Yaskawa INFORM job: turntable_planes_program.JBI

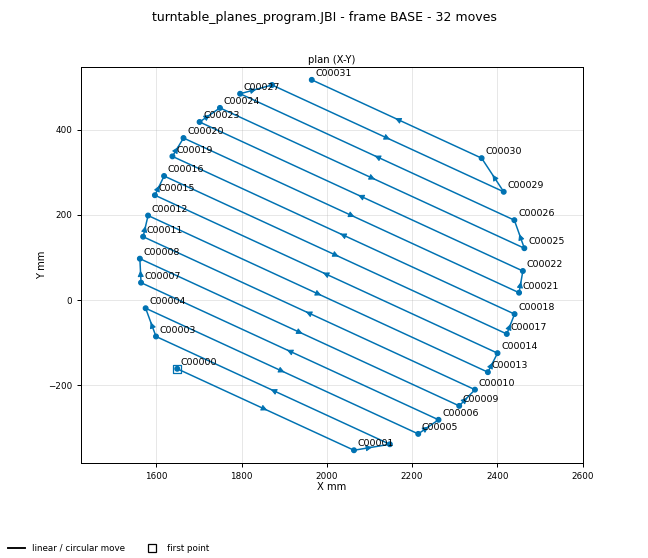
[picture p0: tool path of turntable_planes_program.JBI in frame BASE, 32 of 34 moves have a stored position in this frame; points joined in program order, loops and branches not executed]
/JOB
//NAME turntable_planes_program
//POS
///NPOS 32,0,32,0,0,0
///TOOL 0
///POSTYPE BASE
///RECTAN
///RCONF 0,0,0,0,0,0,0,0,0,0,0,0,0,0,0,0,0,0,0,0,0,0,0,0
C00000=1648.821901,-161.398281,-672.168400,-175.000000,-5.000000,-5.000000
C00001=2063.630161,-352.610148,-666.258453,-175.000000,-5.000000,-5.000000
C00002=2147.857862,-338.592875,-665.466453,-175.000000,-5.000000,-5.000000
C00003=1599.021883,-85.598993,-672.447453,-175.000000,-5.000000,-5.000000
C00004=1574.696176,-19.329185,-672.760453,-175.000000,-5.000000,-5.000000
C00005=2214.442365,-314.229443,-663.003453,-175.000000,-5.000000,-5.000000
C00006=2262.055456,-281.120864,-660.808453,-175.000000,-5.000000,-5.000000
C00007=1563.938343,40.686315,-672.359453,-175.000000,-5.000000,-5.000000
C00008=1561.162308,97.022491,-672.672453,-175.000000,-5.000000,-5.000000
C00009=2310.665703,-248.471939,-661.270453,-175.000000,-5.000000,-5.000000
C00010=2347.574340,-210.428987,-659.728453,-175.000000,-5.000000,-5.000000
C00011=1568.815555,148.551138,-674.488453,-175.000000,-5.000000,-5.000000
C00012=1580.436542,198.250797,-673.419453,-175.000000,-5.000000,-5.000000
C00013=2377.913364,-169.357677,-660.847453,-175.000000,-5.000000,-5.000000
C00014=2400.551212,-124.736398,-661.001453,-175.000000,-5.000000,-5.000000
C00015=1596.436666,245.931830,-668.404453,-175.000000,-5.000000,-5.000000
C00016=1618.017418,291.040392,-663.890453,-175.000000,-5.000000,-5.000000
C00017=2422.299065,-79.704864,-660.760453,-175.000000,-5.000000,-5.000000
C00018=2440.558685,-33.065378,-659.855453,-175.000000,-5.000000,-5.000000
C00019=1637.542101,337.096729,-675.976453,-175.000000,-5.000000,-5.000000
C00020=1663.596438,380.143127,-671.388453,-175.000000,-5.000000,-5.000000
C00021=2451.116220,17.124495,-659.314453,-175.000000,-5.000000,-5.000000
C00022=2460.035439,68.069574,-662.136453,-175.000000,-5.000000,-5.000000
C00023=1701.352386,417.795499,-672.138453,-175.000000,-5.000000,-5.000000
C00024=1749.093527,450.845052,-671.674453,-175.000000,-5.000000,-5.000000
C00025=2463.491181,121.533121,-661.256453,-175.000000,-5.000000,-5.000000
C00026=2440.046386,187.396860,-663.483453,-175.000000,-5.000000,-5.000000
C00027=1796.467772,484.063730,-672.872453,-175.000000,-5.000000,-5.000000
C00028=1871.320142,504.615969,-667.392453,-175.000000,-5.000000,-5.000000
C00029=2415.095866,253.954685,-661.312453,-175.000000,-5.000000,-5.000000
C00030=2363.247179,332.922620,-660.952453,-175.000000,-5.000000,-5.000000
C00031=1964.608666,516.680808,-666.628453,-175.000000,-5.000000,-5.000000
///POSTYPE PULSE
///PULSE
EC00000=250880.0
EC00001=250880.0
EC00002=250880.0
EC00003=250880.0
EC00004=250880.0
EC00005=250880.0
EC00006=250880.0
EC00007=250880.0
EC00008=250880.0
EC00009=250880.0
EC00010=250880.0
EC00011=250880.0
EC00012=250880.0
EC00013=250880.0
EC00014=250880.0
EC00015=250880.0
EC00016=250880.0
EC00017=250880.0
EC00018=250880.0
EC00019=250880.0
EC00020=250880.0
EC00021=250880.0
EC00022=250880.0
EC00023=250880.0
EC00024=250880.0
EC00025=250880.0
EC00026=250880.0
EC00027=250880.0
EC00028=250880.0
EC00029=250880.0
EC00030=250880.0
EC00031=250880.0
//INST
///DATE 2023/08/16 13:45
///ATTR SC,RW,RJ
////FRAME BASE
///GROUP1 RB1,ST1
NOP
MOVJ P009 EX000 VJ=15.00
MOVJ C00000 EC00000 VJ=15.0
CALL JOB:SPYON
MOVL C00001 EC00001 V=150.0
MOVL C00002 EC00002 V=150.0
MOVL C00003 EC00003 V=150.0
MOVL C00004 EC00004 V=150.0
MOVL C00005 EC00005 V=150.0
MOVL C00006 EC00006 V=150.0
MOVL C00007 EC00007 V=150.0
MOVL C00008 EC00008 V=150.0
MOVL C00009 EC00009 V=150.0
MOVL C00010 EC00010 V=150.0
MOVL C00011 EC00011 V=150.0
MOVL C00012 EC00012 V=150.0
MOVL C00013 EC00013 V=150.0
MOVL C00014 EC00014 V=150.0
MOVL C00015 EC00015 V=150.0
MOVL C00016 EC00016 V=150.0
MOVL C00017 EC00017 V=150.0
MOVL C00018 EC00018 V=150.0
MOVL C00019 EC00019 V=150.0
MOVL C00020 EC00020 V=150.0
MOVL C00021 EC00021 V=150.0
MOVL C00022 EC00022 V=150.0
MOVL C00023 EC00023 V=150.0
MOVL C00024 EC00024 V=150.0
MOVL C00025 EC00025 V=150.0
MOVL C00026 EC00026 V=150.0
MOVL C00027 EC00027 V=150.0
MOVL C00028 EC00028 V=150.0
MOVL C00029 EC00029 V=150.0
MOVL C00030 EC00030 V=150.0
MOVL C00031 EC00031 V=150.0
CALL JOB:SPYOF
MOVJ P009 VJ=15.00
END
